FUNCTION_BLOCK FbTOF (* Таймер с задержкой на выключение. *)
  (* Standard: 61499-1; Description: Таймер с задержкой на выключение. Simple FB with one algorithm *)
  (* Version 2.2, 2026-03-14, VA, LIB_PLC *)
  (* Documentation:
  // Таймер с задержкой на выключение. //          DbTOF //    +----------------+ //    |     FbTOF      | // ->-|In           Out|->- //   -|TimeDelayOff    | //   -|Ts_ms           | //    +----------------+  // Применение. // // Блок может применятся как фильтр дребезга контактов и как расширитель им-пульсов. // Временная характеристика. // //  In //  ^ //  |     TimeDelayOff          TimeDelayOff //  |       |<--->|               |<--->| // 1|   *****     |     ***** *** *     | //  |   *   *     |     *   * * * *     | // 0*****---*************---***-*************----> t[s] // //  Out //  ^ //  |     TimeDelayOff          TimeDelayOff //  |       |<--->|               |<--->| // 1|   ***********     ***************** //  |   *         *     *               * // 0*****---------*******---------------*****----> t[s]
  *)
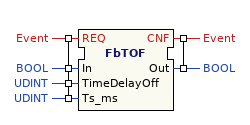
  EVENT_INPUT
    REQ WITH In, TimeDelayOff, Ts_ms; (* Normal Execution Request *)
  END_EVENT
  EVENT_OUTPUT
    CNF WITH Out; (* Execution Confirmation *)
  END_EVENT
  VAR_INPUT
    In : BOOL := FALSE; (* Вход таймера. *)
    TimeDelayOff : UDINT := 5000; (* Время задержки выключения [мс]. *)
    Ts_ms : UDINT := 100; (* Шаг дискретизации по времени [мс]. *)
  END_VAR
  VAR_OUTPUT
    Out : BOOL := FALSE; (* Выход таймера. *)
  END_VAR
  VAR
    Timer1 : UDINT := 0; (* Текущее время таймер1 [мс]. *)
  END_VAR
  EC_STATES
    REQ : REQ -> CNF;
  END_STATES
  ALGORITHM REQ IN ST:
IF (TimeDelayOff > 0) THEN // Таймер включен.
	IF (In) THEN // На входе 1 то на выходе тоже 1.
		Out := TRUE;
		Timer1 := 0;
	ELSE // Если на входе 0.
		IF (Out) THEN // На выходе 1.
			IF (Timer1 >= TimeDelayOff) THEN // Задержка включения закончилась.
				Out := FALSE;
				Timer1 := 0;
			ELSE // Задержка включения активна.
				Out := TRUE;
				Timer1 := Timer1 + Ts_ms;
			END_IF;
		ELSE // На выходе 0.
			Out := FALSE;
			Timer1 := 0;
		END_IF;
	END_IF;
ELSE // Таймер выключен.
	Out := In;
	Timer1 := 0;
END_IF;

// @COPYLEFT ALL WRONGS RESERVED :)
// Author: VA
// Contacts: DIY.PLC.314@gmail.com
// Date start LIB_PLC: 2014
// License: GNU GPL-2.0-or-later
// https://www.gnu.org/licenses/old-licenses/gpl-2.0.html
// https://www.youtube.com/watch?v=n1F_MfLRlX0
// https://www.youtube.com/@DIY_PLC
// https://github.com/DIYPLC/LIB_PLC
// https://oshwlab.com/diy.plc.314/PLC_HW1_SW1
// https://3dtoday.ru/3d-models/mechanical-parts/body/korpus-na-din-reiku
// https://t.me/DIY_PLC
  END_ALGORITHM
END_FUNCTION_BLOCK
